INTERFACE PUBLIC I_AxisJogger

END_INTERFACE

(* stored: Version 1.1.0.1, ProductVersion 3.1.4024.12
   Itf I_AxisJogger: Id {48e41886-d123-0619-3a5c-20d6a492c4b8} *)
